// TIA Portal V19 export
DATA_BLOCK "RECIRCULATION DB"   // DB63
{ S7_Optimized_Access := 'TRUE' }
// stored: MemoryReserve 100
   VAR RETAIN
      MFG : Struct
         START : Bool;
         STOP : Bool;
         PAUSE : Bool;
         BUFF : Int;
      END_STRUCT;
      PREMIXING : Struct
         START : Bool;
         STOP : Bool;
         PAUSE : Bool;
         BUFF : Int;
      END_STRUCT;
      "MFG RECIRCULATION TIME SET" : Int;
   END_VAR
   VAR
      "MFG RECIRCULATION TIME PV" : Int;
   END_VAR
   VAR RETAIN
      "PREMIXING RECIRCULATION TIME SET" : Int;
   END_VAR
   VAR
      "PREMIXING RECIRCULATION TIME PV" : Int;
   END_VAR
BEGIN
END_DATA_BLOCK
